// TIA Portal V21 export
FUNCTION "TEMP" : Void   // FC14, LAD
{ S7_Optimized_Access := 'TRUE' }
// stored: SetENOAutomatically false
   VAR_INPUT
      AI : Int;
      OFFSET : Real;
   END_VAR
   VAR_OUTPUT
      OUT : Real;
   END_VAR
   VAR_TEMP
      TEMP1 : Real;
      temp2 : Real;
   END_VAR
BEGIN

REGION Network 1
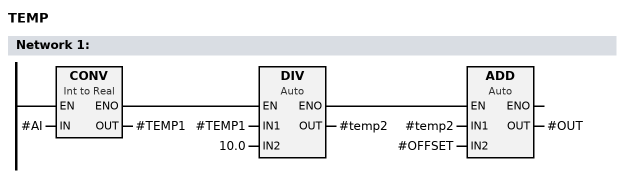
   RUNG wire#powerrail
      { S7_Templates := "[SrcType := Int, DestType := Real]" } Convert(in := #AI, out => #TEMP1)
      Div(in1 := #TEMP1, in2 := 10.0, out => #temp2)
      Add(in1 := #temp2, in2 := #OFFSET, out => #OUT)
   END_RUNG
   // the same network as SCL:
   #TEMP1 := INT_TO_REAL(#AI);
   #temp2 := #TEMP1 / 10.0;
   #OUT := #temp2 + #OFFSET;
END_REGION
END_FUNCTION
